FUNCTION_BLOCK W4W2
  (* Standard: 61499-2 *)
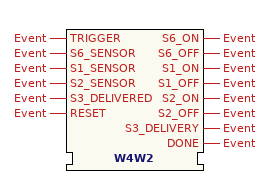
  EVENT_INPUT
    TRIGGER;
    S6_SENSOR;
    S1_SENSOR;
    S2_SENSOR;
    S3_DELIVERED;
    RESET;
  END_EVENT
  EVENT_OUTPUT
    S6_ON;
    S6_OFF;
    S1_ON;
    S1_OFF;
    S2_ON;
    S2_OFF;
    S3_DELIVERY;
    DONE;
  END_EVENT
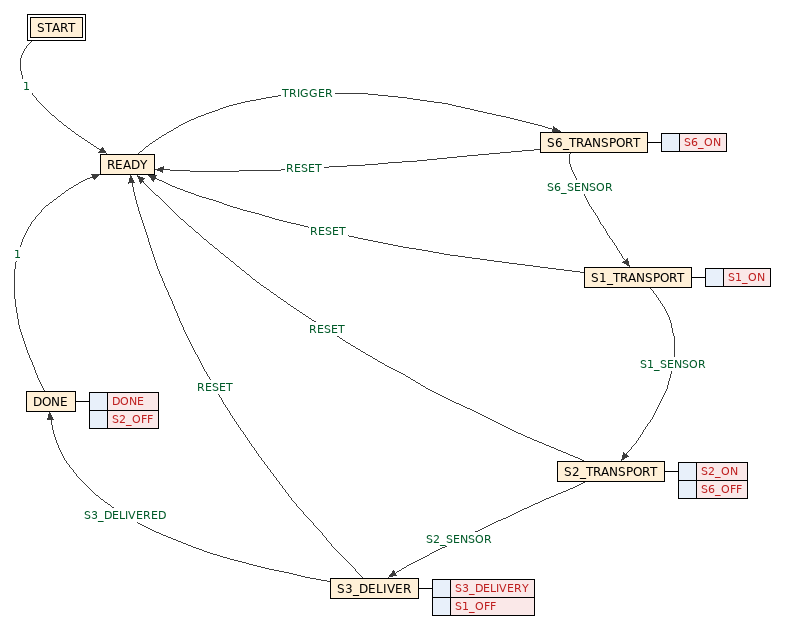
  EC_STATES
    START;
    S6_TRANSPORT : -> S6_ON;
    S1_TRANSPORT : -> S1_ON;
    S3_DELIVER : -> S3_DELIVERY, -> S1_OFF;
    DONE : -> DONE, -> S2_OFF;
    READY;
    S2_TRANSPORT : -> S2_ON, -> S6_OFF;
  END_STATES
  EC_TRANSITIONS
    START TO READY := 1;
    S6_TRANSPORT TO S1_TRANSPORT := S6_SENSOR;
    S3_DELIVER TO DONE := S3_DELIVERED;
    READY TO S6_TRANSPORT := TRIGGER;
    DONE TO READY := 1;
    S1_TRANSPORT TO S2_TRANSPORT := S1_SENSOR;
    S2_TRANSPORT TO S3_DELIVER := S2_SENSOR;
    S6_TRANSPORT TO READY := RESET;
    S1_TRANSPORT TO READY := RESET;
    S2_TRANSPORT TO READY := RESET;
    S3_DELIVER TO READY := RESET;
  END_TRANSITIONS
  ALGORITHM INIT IN ST:

  END_ALGORITHM
  ALGORITHM REQ IN ST:

  END_ALGORITHM
END_FUNCTION_BLOCK
